TYPE SC_BUSY_FirstFloor :
(
	enum_member := 0
);
END_TYPE

(* stored: Version 1.1.0.1, ProductVersion 3.1.4024.2
   DUT SC_BUSY_FirstFloor: Id {f0336001-cfb1-42ab-b3de-eac46dbdd795} *)
